// TIA Portal V21 export
FUNCTION "AmbiguousTarget" : Void   // FC, LAD
// stored: SetENOAutomatically false
BEGIN
END_FUNCTION
